FUNCTION TN_SC_SHADOW_ATTR : BYTE
VAR_INPUT
	Iby_ATTR : BYTE;
END_VAR

(*
version 1.0		10. mai 2010
programmer		ks
tested by		ks

TN_SC_SHADOW_ATTR berechnet aus einem normalen einem abgedunkelten Farbcode
*)

(* Background Farbe auf Schwarz ändern      *)
(* und dunkle Fordergrundfarben einschalten *)  
TN_SC_SHADOW_ATTR := ((Iby_ATTR AND BYTE#2#11110000) OR BYTE#2#00001000);

(* revision history
ks	10. mai. 2010	rev 1.0
	original version
*)

END_FUNCTION

(* stored: Version 1.1.0.1, ProductVersion 3.1.4024.0
   POU TN_SC_SHADOW_ATTR: Id {dc3d62d5-c4e2-4645-8499-825e676c915a}, SpecialFunc None *)
